// TIA Portal project "CompMC_TestProject" (V16)
// REr: Test project 1, RVS reiniging simpel

(* hardware
DEVICE "S71500/ET200MP station_1"  S7-1500 station
   slot 0: "Rail_0"  Rack  6ES7 590-1***0-0AA0
   slot 1: "PLC_1"  CPU 1513F-1 PN  6ES7 513-1FL02-0AB0  V2.8
      slot 3: "CPU display_1"  6ES7591-1AA00-0AA0
      slot 32768: "PROFINET interface_1"  X1
         slot 32769: "Port_1"  X1 P1
         slot 32770: "Port_2"  X1 P2
      slot 34817: "Virtual CP interface port_1"  Virtual CP interface port  Virtual CP interface port
   slot 2: "DI 16x24VDC / DQ 16x24VDC/0.5A BA_1"  DI 16x24VDC/DQ 16x24VDC/0.5A BA  6ES7 523-1BL00-0AA0  V1.1
*)

// ===== PLC "PLC_1"  CPU 1513F-1 PN =====

VAR_GLOBAL   // PLC tag table "Default tag table"
   "Tag_1" AT %M0.0 : Bool;
   "Var X" AT %MW100 : Word;
   "Alarm_1" AT %M102.0 : Bool;
   "Alarm_2" AT %M102.1 : Bool;
   "Alarm_3" AT %M102.2 : Bool;
   "Alarm_4" AT %M102.3 : Bool;
   "Result_as_Expected" AT %M103.0 : Bool;
   "X" AT %MW500 : Word;   // Variable X
   "Xnot10" AT %M400.0 : Bool;   // X != 10
   "Xnot12" AT %M400.1 : Bool;   // X != 12
   "Xnot15" AT %M400.2 : Bool;   // X != 15
   "Xnot20" AT %M400.3 : Bool;   // X != 20
   "NOK" AT %M400.7 : Bool;   // Result NOK
END_VAR

VAR_GLOBAL   // PLC tag table "InOut"
   "Ib_VlvLiq1Opened" AT %I0.0 : Bool;   // Valve liquid 1 openend
   "Ib_VlvLiq1Closed" AT %I0.1 : Bool;   // Valve liquid 1 closed
   "Ib_VlvLiq2Opened" AT %I0.2 : Bool;   // Valve liquid 2 opened
   "Ib_VlvLiq2Closed" AT %I0.3 : Bool;   // Valve liquid 2 closed
   "Ib_VlvDrnOpened" AT %I0.4 : Bool;   // Valve drain opened
   "Ib_VlvDrnClosed" AT %I0.5 : Bool;   // Valve drain closed
   "Ib_LvlContEmpty" AT %I0.6 : Bool;   // Level container empty
   "Ib_LvlContFull" AT %I0.7 : Bool;   // Level container full
   "Ib_PBFillLiq1" AT %I1.0 : Bool;   // Pushbutton fill container with liquid 1
   "Ib_PBFillLiq2" AT %I1.1 : Bool;   // Pushbutton fill container with liquid 2
   "Ib_PBEmptyCont" AT %I1.2 : Bool;   // Pushbutton empty container
   "Qb_VlvLiq1Open" AT %Q0.0 : Bool;   // Valve liquid 1 move open
   "Qb_VlvLiq2Open" AT %Q0.1 : Bool;   // Valve liquid 2 move open
   "Qb_VlvDrnOpen" AT %Q0.2 : Bool;   // Valve drain move open
   "Ib_PBStart" AT %I1.3 : Bool;   // Pushbutton start
   "Ib_PBStop" AT %I1.4 : Bool;   // Pushbutton stop
   "Ib_PBReset" AT %I1.5 : Bool;   // Pushbutton reset
END_VAR

VAR_GLOBAL CONSTANT   // PLC tag table "Open Library"
   "Modes.Auto" : Int := 1;
   "Modes.Manual" : Int := 2;
   "Modes.Independent" : Int := 10;
   "Modes.Stop" : Int := 0;
   "HMI.Status.Stopped" : Int := 0;
   "HMI.Status.Estop" : Int := 1;
   "HMI.Status.Error" : Int := 2;
   "HMI.Status.ForwardWork" : Int := 3;
   "HMI.Status.ReverseHome" : Int := 4;
   "HMI.Status.OnForwardWork" : Int := 5;
   "HMI.Status.OnReverseHome" : Int := 6;
   "IoScaling.S7Analog.Default.iRawMax" : Int := 27648;
   "IoScaling.S7Analog.Default.iRawMin" : Int := 0;
   "IoScaling.S7Analog.Default.bSwapBytes" : Bool := false;
   "IoScaling.S7Analog.+-V/mA.iRawMax" : Int := 27648;
   "IoScaling.S7Analog.+-V/mA.iRawMin" : Int := -27648;
   "IoScaling.S7Analog.Types.Default" : Int := 0;
   "IoScaling.S7Analog.Pt100.iRawMax" : Int := 8500;
   "IoScaling.S7Analog.Pt100.iRawMin" : Int := -2000;
   "IoScaling.S7Analog.Pt100.Climate.iRawMax" : Int := 13000;
   "IoScaling.S7Analog.Pt100.Climate.iRawMin" : Int := -12000;
   "IoScaling.S7Analog.Ni100.iRawMax" : Int := 2500;
   "IoScaling.S7Analog.Ni100.iRawMin" : Int := -600;
   "IoScaling.S7Analog.Ni100.Climate.iRawMax" : Int := 25000;
   "IoScaling.S7Analog.Ni100.Climate.iRawMin" : Int := -6000;
   "IoScaling.S7Analog.Types.+-V/mA" : Int := 1;
   "IoScaling.S7Analog.Types.Pt100" : Int := 2;
   "IoScaling.S7Analog.Types.Pt100.Climate" : Int := 3;
   "IoScaling.S7Analog.Types.Ni100" : Int := 4;
   "IoScaling.S7Analog.Types.Ni100.Climate" : Int := 5;
   "IoScaling.S7Analog.Pt100.rScaledMax" : Real := 850.0;
   "IoScaling.S7Analog.Pt100.rScaledMin" : Real := -200.0;
   "IoScaling.S7Analog.Pt100.Climate.rScaledMax" : Real := 130.0;
   "IoScaling.S7Analog.Pt100.Climate.rScaledMin" : Real := -120.0;
   "IoScaling.S7Analog.Ni100.rScaledMax" : Real := 250.0;
   "IoScaling.S7Analog.Ni100.rScaledMin" : Real := -60.0;
   "IoScaling.S7Analog.Ni100.Climate.rScaledMax" : Real := 250.0;
   "IoScaling.S7Analog.Ni100.Climate.rScaledMin" : Real := -60.0;
   "IoScaling.S7Analog.150Ohms.rScaledMax" : Real := 150.0;
   "IoScaling.S7Analog.150Ohms.rScaledMin" : Real := 0.0;
   "IoScaling.S7Analog.300Ohms.rScaledMax" : Real := 300.0;
   "IoScaling.S7Analog.300Ohms.rScaledMin" : Real := 0.0;
   "IoScaling.S7Analog.600Ohms.rScaledMax" : Real := 600.0;
   "IoScaling.S7Analog.600Ohms.rScaledMin" : Real := 0.0;
   "Estop.MinSetPoint" : Int := 0;
   "Estop.MaxSetPoint" : Int := 1;
   "Estop.HMISetPoint" : Int := 2;
   "Modes.PID.Inactive" : Int := 0;
   "Modes.PID.Pretuning" : Int := 1;
   "Modes.PID.FineTuning" : Int := 2;
   "Modes.PID.AutoMode" : Int := 3;
   "Modes.PID.ManualMode" : Int := 4;
   "HMI.Status.Generic1" : Int := 101;
   "HMI.Status.Generic2" : Int := 102;
   "HMI.Status.Generic3" : Int := 103;
   "HMI.Status.Generic4" : Int := 104;
   "HMI.Status.Generic5" : Int := 105;
   "HMI.Status.GenericNone" : Int := 100;
   "HMI.Status.Generic6" : Int := 106;
   "DataTypes.rMaxReal" : Real := 3.402823e38;
   "DataTypes.rMinReal" : Real := -3.402823e38;
   "DataTypes.iMaxInt" : Int := 32767;
   "DataTypes.iMinInt" : Int := -32768;
   "Handshakes.iSize" : Int := 5;
   "SoftStarter.Types.3RW30" : Int := 30;
   "SoftStarter.Types.3RW40" : Int := 40;
   "Simocode.Types.OverloadRelay" : Int := 0;
   "Simocode.Types.DirectStarter" : Int := 1;
   "Simocode.Types.ReversingStarter" : Int := 2;
   "SoftStarter.HMI.Status.RampDown" : Int := 5;
   "SoftStarter.HMI.Status.On" : Int := 4;
   "SoftStarter.HMI.Status.RampUp" : Int := 3;
   "SoftStarter.HMI.Status.EStop" : Int := 1;
   "SoftStarter.HMI.Status.Off" : Int := 0;
   "SoftStarter.HMI.Status.Error" : Int := 2;
   "FIFO.iQueueSize" : Int := 5;
   "FIFO.iQueueDisabled" : Int := -1;
   "TotalizerTimeUnits.MILLISECONDS" : Int := 0;
   "TotalizerTimeUnits.SECONDS" : Int := 1;
   "TotalizerTimeUnits.MINUTES" : Int := 2;
   "TotalizerTimeUnits.HOURS" : Int := 3;
   "TotalizerTimeUnits.DAYS" : Int := 4;
   "HMI.Status.SimulatedForwardWork" : Int := 7;
   "HMI.Status.SimulatedOnForwardWork" : Int := 9;
   "HMI.Status.SimulatedReverseHome" : Int := 8;
   "HMI.Status.SimulatedOnReverseHome" : Int := 10;
   "Ramp.Continuous" : Int := 0;
   "Ramp.Timed" : Int := 1;
END_VAR

// folder: Open Library V15/Data Types/Error

TYPE "udtError_Valve"
VERSION : 0.1
   STRUCT
      NoHomeFeedback : Bool;   // Home position feedback not active
      NoWorkFeedback : Bool;   // Work position feedback not active
      HomeFeedbackStillActive : Bool;   // Home position feedback still active
      WorkFeedbackStillActive : Bool;   // Work position feedback still active
   END_STRUCT;
END_TYPE

// folder: Open Library V15/Data Types/HMI

TYPE "udtHMI_ValveControl"
VERSION : 0.1
   STRUCT
      iMode : Int;   // Current mode
      iErrorCode : Int;   // Error code
      iStatus : Int;   // Status for HMI display
      bPB_ResetError : Bool;   // PB Reset block errors
      bPB_Home : Bool;   // PB Move to home in manual mode
      bPB_Work : Bool;   // PB Move to work in manual mode
      bPBEN_ResetError : Bool;   // PB Reset error enabled
      bPBEN_Home : Bool;   // PB Home enabled
      bPBEN_Work : Bool;   // PB Work enabled
      bHomeOn : Bool;   // Home command is on
      bWorkOn : Bool;   // Work command is on
      bSignalHome : Bool;   // Home feedback
      bSignalWork : Bool;   // Work feedback
      bError : Bool;   // Error status
      bInterlock : Bool;   // Valve interlocked
   END_STRUCT;
END_TYPE

// folder: (top level)

DATA_BLOCK "Program Logic_DB"   // DB2
{ S7_Optimized_Access := 'TRUE' }
VERSION : 0.1
// stored: InstanceOfName Program Logic
"Program Logic"
BEGIN
END_DATA_BLOCK

DATA_BLOCK "DB_HMI"   // DB3
{ S7_Optimized_Access := 'TRUE' }
VERSION : 0.1
   VAR
      VlvLiq1 : "udtHMI_ValveControl";
      VlvLiq2 : "udtHMI_ValveControl";
      VlvDrn : "udtHMI_ValveControl";
   END_VAR
BEGIN
END_DATA_BLOCK

DATA_BLOCK "DB_ProgramLogic"   // DB4
{ S7_Optimized_Access := 'TRUE' }
VERSION : 0.1
   VAR
      VlvLiq1_Open : Bool;
      VlvLiq2_Open : Bool;
      VlvDrn_Open : Bool;
   END_VAR
BEGIN
END_DATA_BLOCK

DATA_BLOCK "Valve Drain_DB"   // DB7
{ S7_Optimized_Access := 'TRUE' }
VERSION : 0.1
// stored: InstanceOfName Valve Drain
"Valve Drain"
BEGIN
END_DATA_BLOCK

DATA_BLOCK "Valve Liquid 1_DB"   // DB8
{ S7_Optimized_Access := 'TRUE' }
VERSION : 0.1
// stored: InstanceOfName Valve Liquid 1
"Valve Liquid 1"
BEGIN
END_DATA_BLOCK

DATA_BLOCK "Valve Liquid 2_DB"   // DB9
{ S7_Optimized_Access := 'TRUE' }
VERSION : 0.1
// stored: InstanceOfName Valve Liquid 2
"Valve Liquid 2"
BEGIN
END_DATA_BLOCK

FUNCTION_BLOCK "Valve Liquid 1"   // FB2, FBD
{ S7_Optimized_Access := 'TRUE' }
VERSION : 0.1
   VAR
      VlvLiq1 : "fbValve_Solenoid";
   END_VAR
BEGIN

REGION Network 1
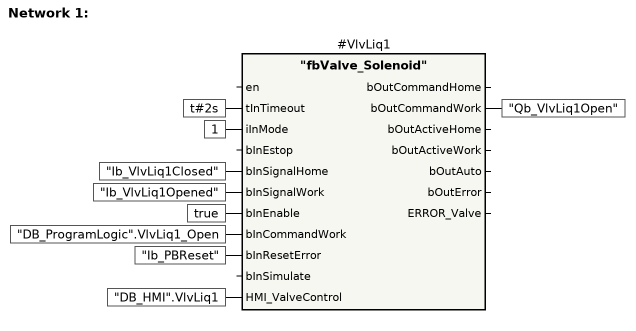
   #VlvLiq1(tInTimeout := t#2s,   // "fbValve_Solenoid"
            iInMode := 1,
            bInSignalHome := "Ib_VlvLiq1Closed",
            bInSignalWork := "Ib_VlvLiq1Opened",
            bInEnable := true,
            bInCommandWork := "DB_ProgramLogic".VlvLiq1_Open,
            bInResetError := "Ib_PBReset",
            HMI_ValveControl := "DB_HMI".VlvLiq1,
            bOutCommandWork => "Qb_VlvLiq1Open");
END_REGION
END_FUNCTION_BLOCK

FUNCTION_BLOCK "Valve Liquid 2"   // FB3, FBD
{ S7_Optimized_Access := 'TRUE' }
VERSION : 0.1
   VAR
      VlvLiq2 : "fbValve_Solenoid";
   END_VAR
BEGIN

REGION Network 1
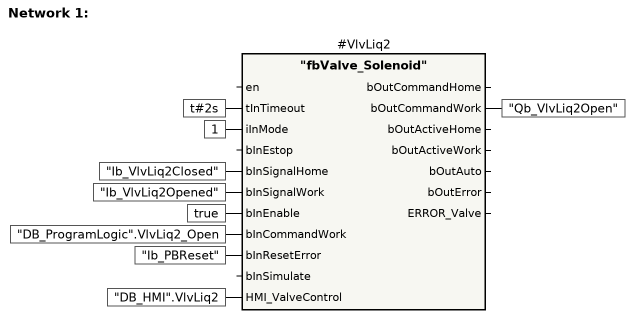
   #VlvLiq2(tInTimeout := t#2s,   // "fbValve_Solenoid"
            iInMode := 1,
            bInSignalHome := "Ib_VlvLiq2Closed",
            bInSignalWork := "Ib_VlvLiq2Opened",
            bInEnable := true,
            bInCommandWork := "DB_ProgramLogic".VlvLiq2_Open,
            bInResetError := "Ib_PBReset",
            HMI_ValveControl := "DB_HMI".VlvLiq2,
            bOutCommandWork => "Qb_VlvLiq2Open");
END_REGION
END_FUNCTION_BLOCK

FUNCTION_BLOCK "Valve Drain"   // FB4, FBD
{ S7_Optimized_Access := 'TRUE' }
VERSION : 0.1
   VAR
      VlvDrn : "fbValve_Solenoid";
   END_VAR
BEGIN

REGION Network 1
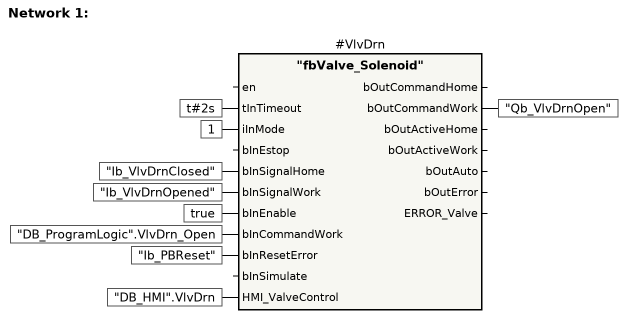
   #VlvDrn(tInTimeout := t#2s,   // "fbValve_Solenoid"
           iInMode := 1,
           bInSignalHome := "Ib_VlvDrnClosed",
           bInSignalWork := "Ib_VlvDrnOpened",
           bInEnable := true,
           bInCommandWork := "DB_ProgramLogic".VlvDrn_Open,
           bInResetError := "Ib_PBReset",
           HMI_ValveControl := "DB_HMI".VlvDrn,
           bOutCommandWork => "Qb_VlvDrnOpen");
END_REGION
END_FUNCTION_BLOCK

FUNCTION_BLOCK "Program Logic"   // FB5, FBD
{ S7_Optimized_Access := 'TRUE' }
VERSION : 0.1
   VAR
      StepSeq : "fbStepSequencer";
      CurrentStep : Int;
      NextStep : Int;
      StepDone : Bool;
   END_VAR
   VAR_TEMP   // added for the SCL form of the ladder/FBD networks
      _w1 : Bool;
   END_VAR
BEGIN

REGION Network 1: 0 -- Idle
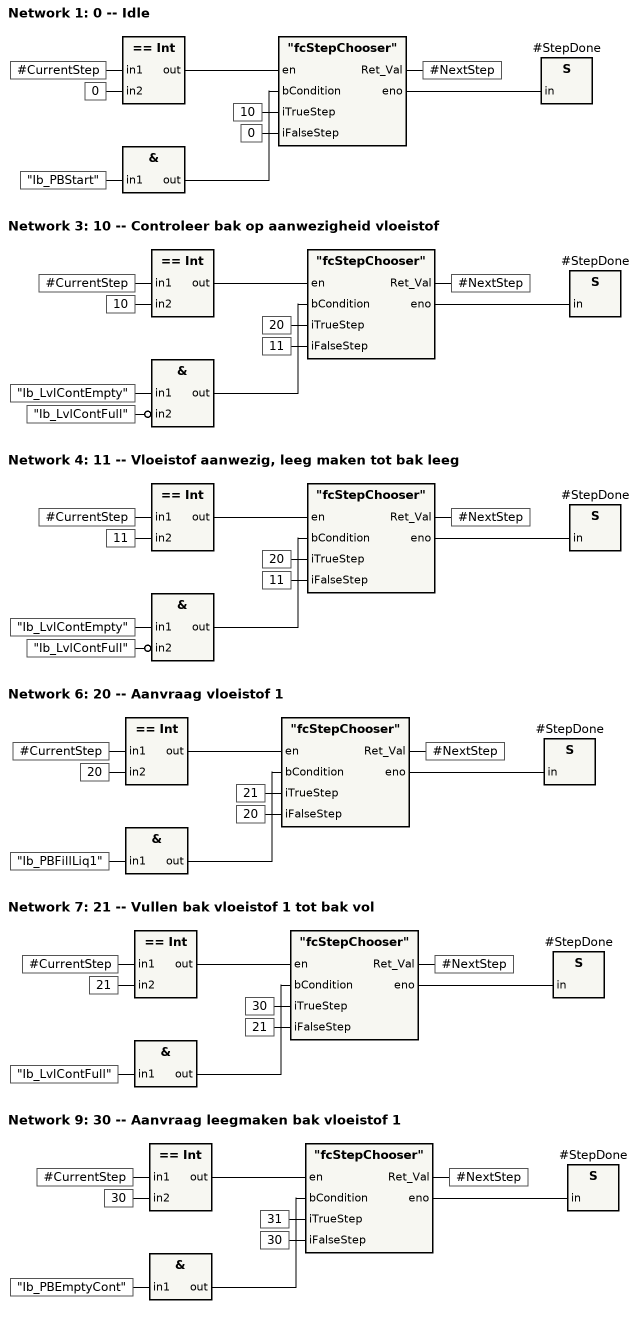
   #NextStep := "fcStepChooser"(EN := #CurrentStep = 0,
                           bCondition := "Ib_PBStart",
                           iTrueStep := 10,
                           iFalseStep := 0,
                           ENO => #_w1);
   IF #_w1 THEN #StepDone := TRUE; END_IF;
END_REGION

REGION Network 3: 10 -- Controleer bak op aanwezigheid vloeistof
   // vloeistof aanwezig 10->11
   // geen vloeistof aanwezig 10->20
   #NextStep := "fcStepChooser"(EN := #CurrentStep = 10,
                           bCondition := "Ib_LvlContEmpty" AND NOT "Ib_LvlContFull",
                           iTrueStep := 20,
                           iFalseStep := 11,
                           ENO => #_w1);
   IF #_w1 THEN #StepDone := TRUE; END_IF;
END_REGION

REGION Network 4: 11 -- Vloeistof aanwezig, leeg maken tot bak leeg
   #NextStep := "fcStepChooser"(EN := #CurrentStep = 11,
                           bCondition := "Ib_LvlContEmpty" AND NOT "Ib_LvlContFull",
                           iTrueStep := 20,
                           iFalseStep := 11,
                           ENO => #_w1);
   IF #_w1 THEN #StepDone := TRUE; END_IF;
END_REGION

REGION Network 6: 20 -- Aanvraag vloeistof 1
   #NextStep := "fcStepChooser"(EN := #CurrentStep = 20,
                           bCondition := "Ib_PBFillLiq1",
                           iTrueStep := 21,
                           iFalseStep := 20,
                           ENO => #_w1);
   IF #_w1 THEN #StepDone := TRUE; END_IF;
END_REGION

REGION Network 7: 21 -- Vullen bak vloeistof 1 tot bak vol
   #NextStep := "fcStepChooser"(EN := #CurrentStep = 21,
                           bCondition := "Ib_LvlContFull",
                           iTrueStep := 30,
                           iFalseStep := 21,
                           ENO => #_w1);
   IF #_w1 THEN #StepDone := TRUE; END_IF;
END_REGION

REGION Network 9: 30 -- Aanvraag leegmaken bak vloeistof 1
   #NextStep := "fcStepChooser"(EN := #CurrentStep = 30,
                           bCondition := "Ib_PBEmptyCont",
                           iTrueStep := 31,
                           iFalseStep := 30,
                           ENO => #_w1);
   IF #_w1 THEN #StepDone := TRUE; END_IF;
END_REGION

REGION Network 10: 31 -- Leeg maken bak vloeistof 1
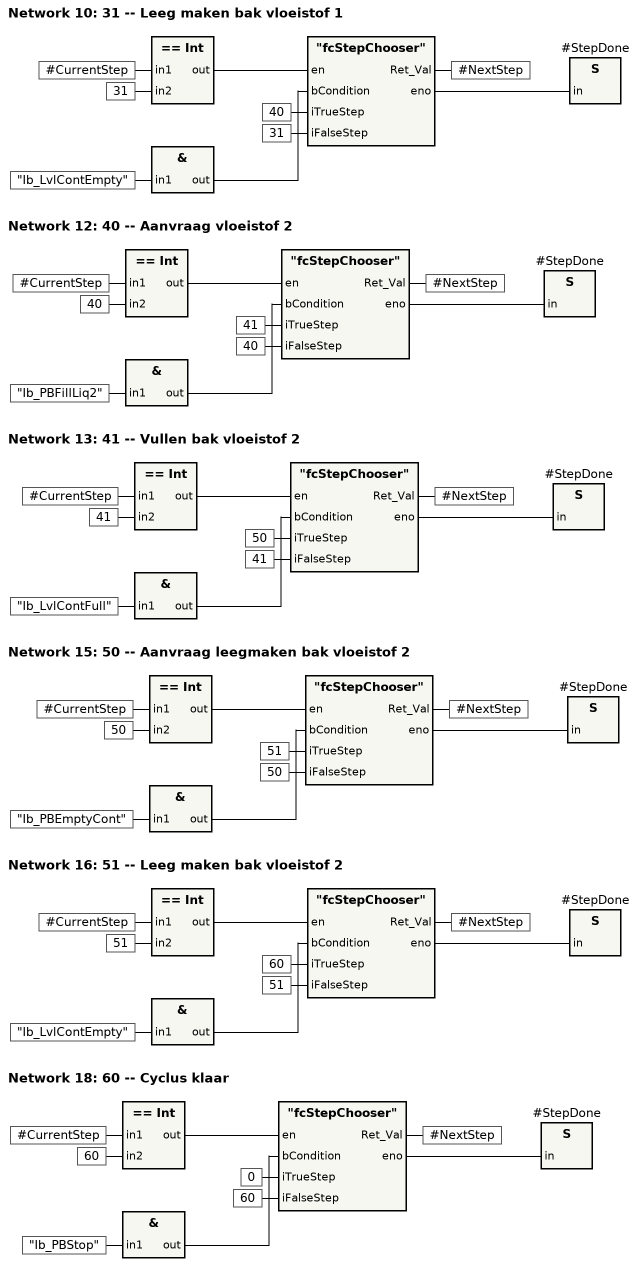
   #NextStep := "fcStepChooser"(EN := #CurrentStep = 31,
                           bCondition := "Ib_LvlContEmpty",
                           iTrueStep := 40,
                           iFalseStep := 31,
                           ENO => #_w1);
   IF #_w1 THEN #StepDone := TRUE; END_IF;
END_REGION

REGION Network 12: 40 -- Aanvraag vloeistof 2
   #NextStep := "fcStepChooser"(EN := #CurrentStep = 40,
                           bCondition := "Ib_PBFillLiq2",
                           iTrueStep := 41,
                           iFalseStep := 40,
                           ENO => #_w1);
   IF #_w1 THEN #StepDone := TRUE; END_IF;
END_REGION

REGION Network 13: 41 -- Vullen bak vloeistof 2
   #NextStep := "fcStepChooser"(EN := #CurrentStep = 41,
                           bCondition := "Ib_LvlContFull",
                           iTrueStep := 50,
                           iFalseStep := 41,
                           ENO => #_w1);
   IF #_w1 THEN #StepDone := TRUE; END_IF;
END_REGION

REGION Network 15: 50 -- Aanvraag leegmaken bak vloeistof 2
   #NextStep := "fcStepChooser"(EN := #CurrentStep = 50,
                           bCondition := "Ib_PBEmptyCont",
                           iTrueStep := 51,
                           iFalseStep := 50,
                           ENO => #_w1);
   IF #_w1 THEN #StepDone := TRUE; END_IF;
END_REGION

REGION Network 16: 51 -- Leeg maken bak vloeistof 2
   #NextStep := "fcStepChooser"(EN := #CurrentStep = 51,
                           bCondition := "Ib_LvlContEmpty",
                           iTrueStep := 60,
                           iFalseStep := 51,
                           ENO => #_w1);
   IF #_w1 THEN #StepDone := TRUE; END_IF;
END_REGION

REGION Network 18: 60 -- Cyclus klaar
   #NextStep := "fcStepChooser"(EN := #CurrentStep = 60,
                           bCondition := "Ib_PBStop",
                           iTrueStep := 0,
                           iFalseStep := 60,
                           ENO => #_w1);
   IF #_w1 THEN #StepDone := TRUE; END_IF;
END_REGION

REGION Network 20: Step Sequencer
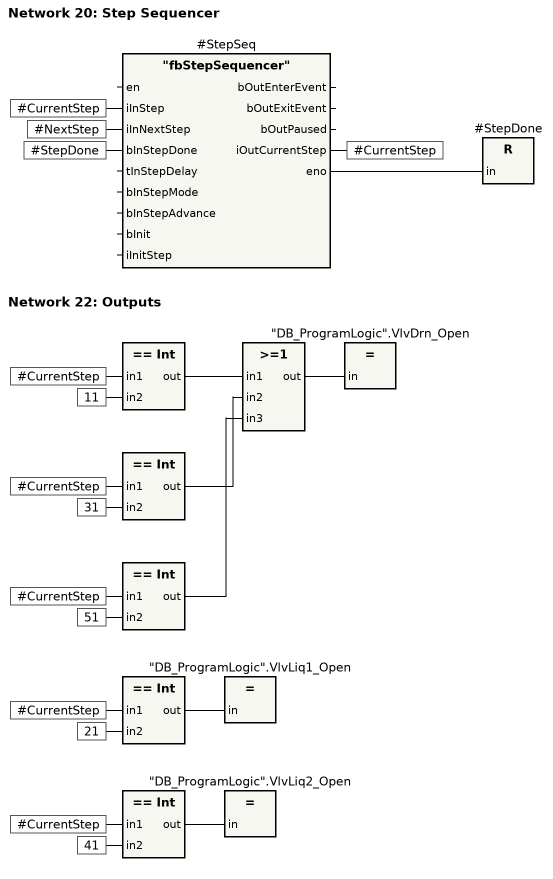
   #StepSeq(iInStep := #CurrentStep,   // "fbStepSequencer"
            iInNextStep := #NextStep,
            bInStepDone := #StepDone,
            iOutCurrentStep => #CurrentStep,
            ENO => #_w1);
   IF #_w1 THEN #StepDone := FALSE; END_IF;
END_REGION

REGION Network 22: Outputs
   "DB_ProgramLogic".VlvDrn_Open := (#CurrentStep = 11) OR (#CurrentStep = 31) OR (#CurrentStep = 51);
   "DB_ProgramLogic".VlvLiq1_Open := #CurrentStep = 21;
   "DB_ProgramLogic".VlvLiq2_Open := #CurrentStep = 41;
END_REGION
END_FUNCTION_BLOCK

ORGANIZATION_BLOCK "Main"   // OB1, FBD, ProgramCycle
TITLE = "Main Program Sweep (Cycle)"
{ S7_Optimized_Access := 'TRUE' }
VERSION : 0.1
   VAR_INPUT
      Initial_Call : Bool;   // Initial call of this OB
      Remanence : Bool;   // =True, if remanent data are available
   END_VAR
BEGIN

REGION Network 1
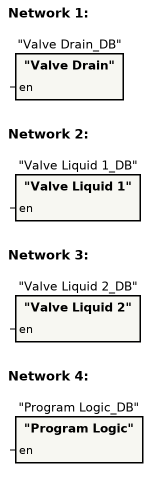
   "Valve Drain_DB"();   // "Valve Drain"
END_REGION

REGION Network 2
   "Valve Liquid 1_DB"();   // "Valve Liquid 1"
END_REGION

REGION Network 3
   "Valve Liquid 2_DB"();   // "Valve Liquid 2"
END_REGION

REGION Network 4
   "Program Logic_DB"();   // "Program Logic"
END_REGION
END_ORGANIZATION_BLOCK

// folder: Open Library V15/Devices

FUNCTION_BLOCK "fbValve_Solenoid"   // FB110, FBD
TITLE = Controls a double- or single-acting valve
{ S7_Optimized_Access := 'TRUE' }
VERSION : 0.1
   VAR_INPUT
      tInTimeout : Time;   // Timeout time for an actuator's feedback to activate before giving a fault
      iInMode : Int;   // Mode Selection
      bInEstop : Bool;   // Estop
      bInSignalHome : Bool;   // Home position feedback
      bInSignalWork : Bool;   // Work position feedback
      bInEnable : Bool;   // Home and Work Enabled
      bInCommandWork : Bool;   // Move to work position in automatic mode
      bInResetError : Bool;   // Reset Error
      bInSimulate : Bool;   // Activate device simulation
   END_VAR
   VAR_OUTPUT
      bOutCommandHome : Bool;   // Home position command
      bOutCommandWork : Bool;   // Work position command
      bOutActiveHome : Bool;   // Valve is in home position
      bOutActiveWork : Bool;   // Valve is in work position
      bOutAuto : Bool;   // Block in auto mode
      bOutError : Bool;   // Error exists
      ERROR_Valve : "udtError_Valve";   // Valve error structure
   END_VAR
   VAR_IN_OUT
      HMI_ValveControl : "udtHMI_ValveControl";   // HMI valve control
   END_VAR
   VAR
      ErrorScroller : "fbErrorScroller";   // Sub-block to handle error scroller
      TON_TimeOut : TON_TIME;   // Timer for Error Timeout
      iLastMode : Int;   // Last mode code
      bNewMode : Bool;   // New mode selected
      bEnableHome : Bool;   // Home position enabled
      bEnableWork : Bool;   // Work position enabled
      bAutoMode : Bool;   // Auto Mode is active
      bManualMode : Bool;   // Manual Mode is active
      bReset : Bool;
      bTON_TimeOut : Bool;
      bPB_Home : Bool;
      bPB_Work : Bool;
      bPB_ResetError : Bool;
   END_VAR
   VAR_TEMP
      tTimeoutElapsed : Time;   // Elapsed time for TON_Timeout
      bTemp : Bool;
   END_VAR
   VAR_TEMP   // added for the SCL form of the ladder/FBD networks
      _w1 : Bool;
      _w2 : Bool;
   END_VAR
BEGIN

REGION Network 1: --------------------------------------------------------- Inputs ------------------------------------------------------------------
END_REGION

REGION Network 2: Read HMI input buttons
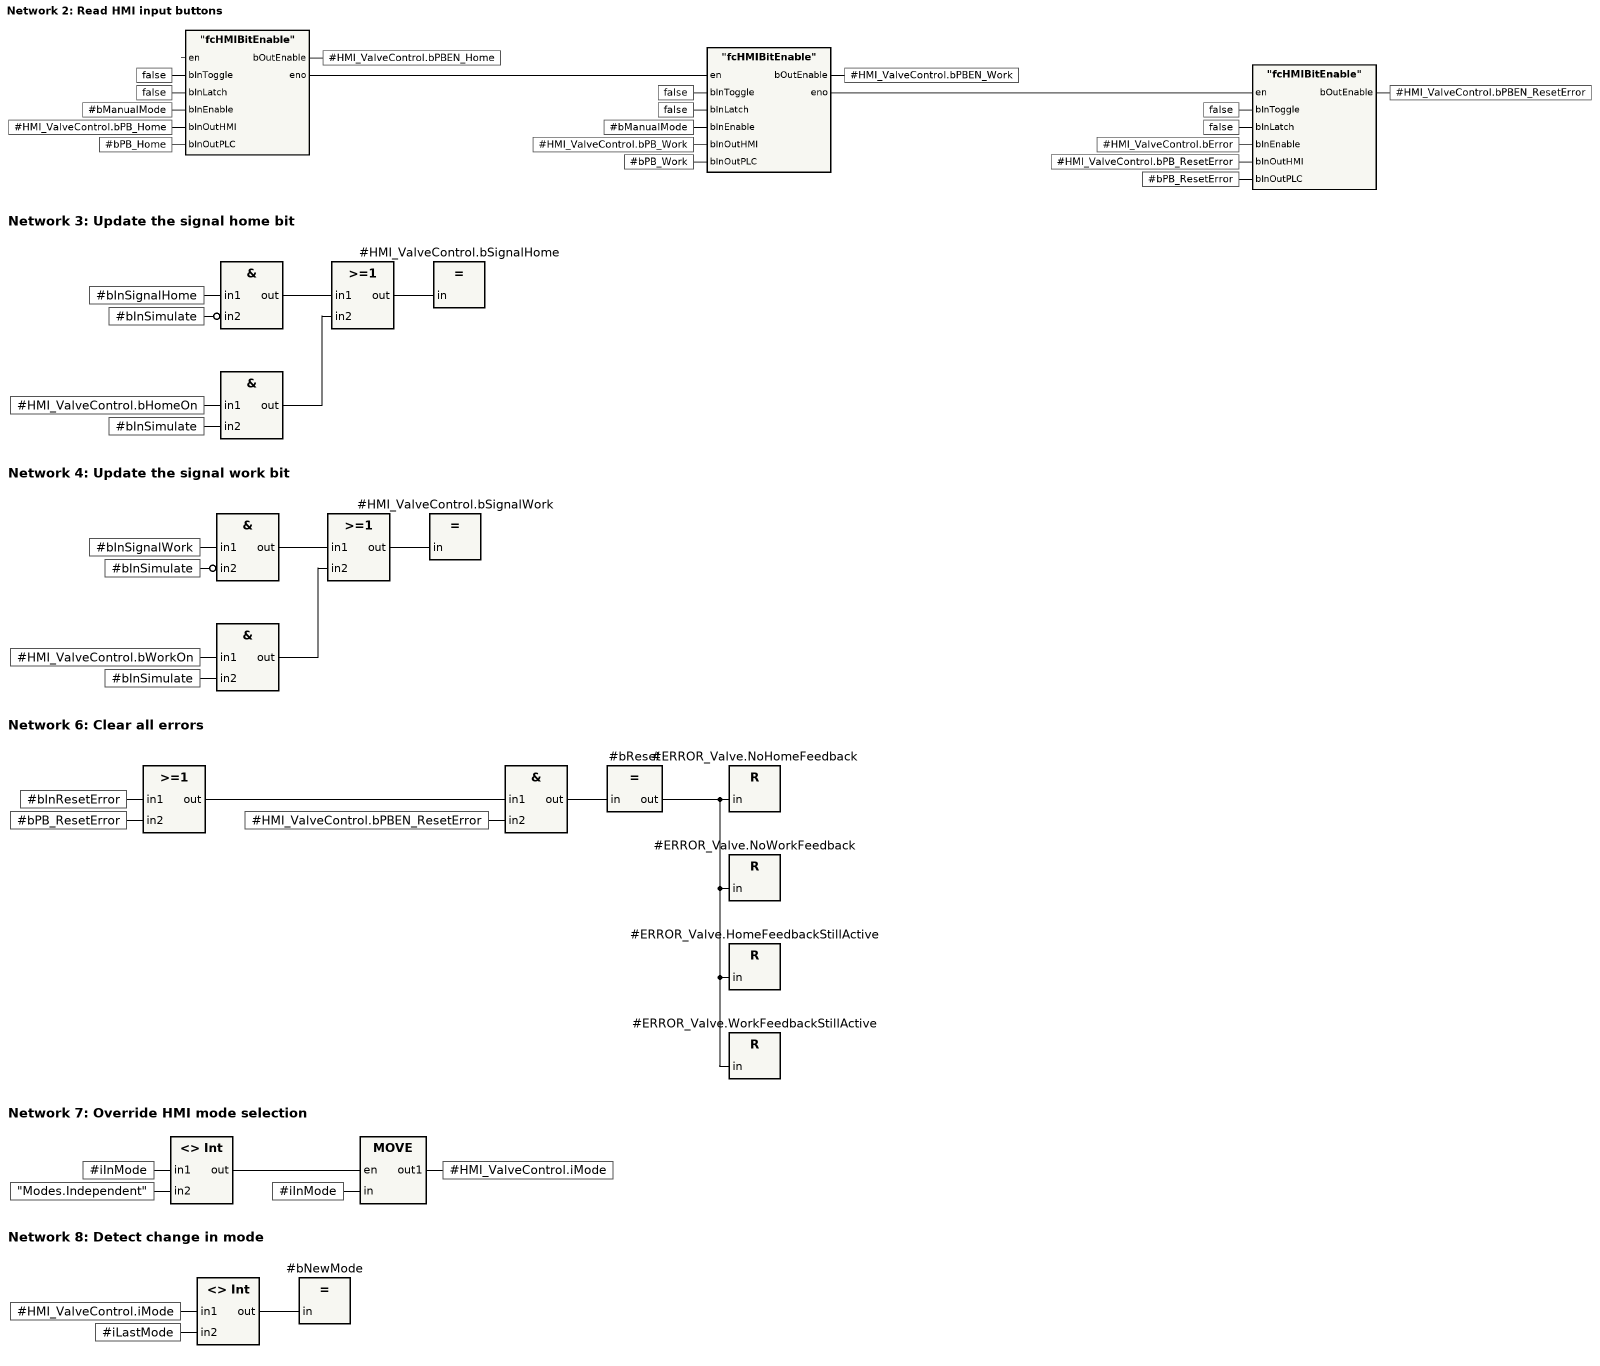
   "fcHMIBitEnable"(bInToggle := false,
                    bInLatch := false,
                    bInEnable := #bManualMode,
                    bInOutHMI := #HMI_ValveControl.bPB_Home,
                    bInOutPLC := #bPB_Home,
                    bOutEnable => #HMI_ValveControl.bPBEN_Home,
                    ENO => #_w1);
   "fcHMIBitEnable"(EN := #_w1,
                    bInToggle := false,
                    bInLatch := false,
                    bInEnable := #bManualMode,
                    bInOutHMI := #HMI_ValveControl.bPB_Work,
                    bInOutPLC := #bPB_Work,
                    bOutEnable => #HMI_ValveControl.bPBEN_Work,
                    ENO => #_w2);
   IF #_w2 THEN
       "fcHMIBitEnable"(bInToggle := false,
                        bInLatch := false,
                        bInEnable := #HMI_ValveControl.bError,
                        bInOutHMI := #HMI_ValveControl.bPB_ResetError,
                        bInOutPLC := #bPB_ResetError,
                        bOutEnable => #HMI_ValveControl.bPBEN_ResetError);
   END_IF;
END_REGION

REGION Network 3: Update the signal home bit
   #HMI_ValveControl.bSignalHome := (#bInSignalHome AND NOT #bInSimulate) OR (#HMI_ValveControl.bHomeOn AND #bInSimulate);
END_REGION

REGION Network 4: Update the signal work bit
   #HMI_ValveControl.bSignalWork := (#bInSignalWork AND NOT #bInSimulate) OR (#HMI_ValveControl.bWorkOn AND #bInSimulate);
END_REGION

REGION Network 5: --------------------------------------------------- Control Logic ------------------------------------------------------------
END_REGION

REGION Network 6: Clear all errors
   #bReset := (#bInResetError OR #bPB_ResetError) AND #HMI_ValveControl.bPBEN_ResetError;
   IF #bReset THEN
       #ERROR_Valve.NoHomeFeedback := FALSE;
       #ERROR_Valve.NoWorkFeedback := FALSE;
       #ERROR_Valve.HomeFeedbackStillActive := FALSE;
       #ERROR_Valve.WorkFeedbackStillActive := FALSE;
   END_IF;
END_REGION

REGION Network 7: Override HMI mode selection
   IF #iInMode <> "Modes.Independent" THEN #HMI_ValveControl.iMode := #iInMode; END_IF;
END_REGION

REGION Network 8: Detect change in mode
   #bNewMode := #HMI_ValveControl.iMode <> #iLastMode;
END_REGION

REGION Network 9: Keep track of last mode
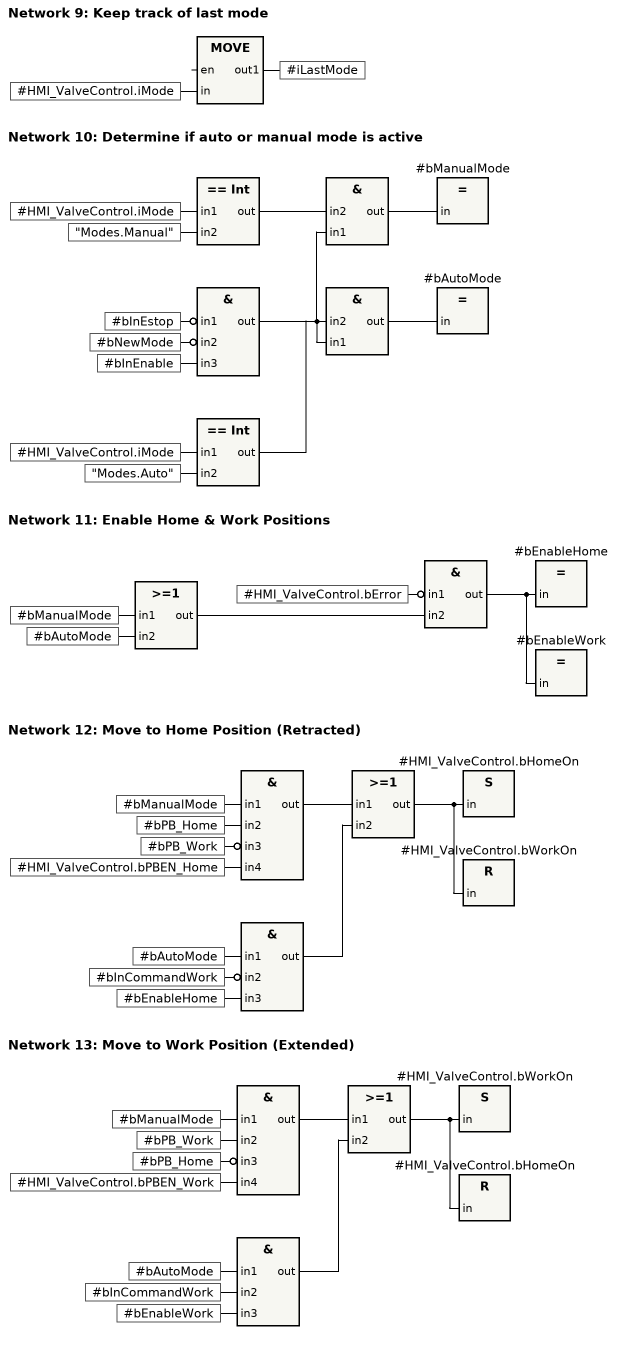
   #iLastMode := #HMI_ValveControl.iMode;
END_REGION

REGION Network 10: Determine if auto or manual mode is active
   #_w1 := NOT #bInEstop AND NOT #bNewMode AND #bInEnable;
   #bManualMode := (#HMI_ValveControl.iMode = "Modes.Manual") AND #_w1;
   #bAutoMode := (#HMI_ValveControl.iMode = "Modes.Auto") AND #_w1;
END_REGION

REGION Network 11: Enable Home & Work Positions
   // IF manual mode AND no estop AND not a new mode AND enabled => 
   // --if no cylinder errors, enable move to Home and Work
   // --enable home and work HMI buttons only in manual mode
   #bEnableHome := NOT #HMI_ValveControl.bError AND (#bManualMode OR #bAutoMode);
   #bEnableWork := #bEnableHome;
END_REGION

REGION Network 12: Move to Home Position (Retracted)
   // IF manual mode and home button is pressed =>
   // --Set close cylinder
   IF (#bManualMode AND #bPB_Home AND NOT #bPB_Work AND #HMI_ValveControl.bPBEN_Home) OR (#bAutoMode AND NOT #bInCommandWork AND #bEnableHome) THEN
       #HMI_ValveControl.bHomeOn := TRUE;
       #HMI_ValveControl.bWorkOn := FALSE;
   END_IF;
END_REGION

REGION Network 13: Move to Work Position (Extended)
   // IF manual mode and work button button is pressed =>
   // --Set open cylinder
   IF (#bManualMode AND #bPB_Work AND NOT #bPB_Home AND #HMI_ValveControl.bPBEN_Work) OR (#bAutoMode AND #bInCommandWork AND #bEnableWork) THEN
       #HMI_ValveControl.bWorkOn := TRUE;
       #HMI_ValveControl.bHomeOn := FALSE;
   END_IF;
END_REGION

REGION Network 14: Reset home on if not enabled
   // IF in auto AND home is not enabled => RESET home command
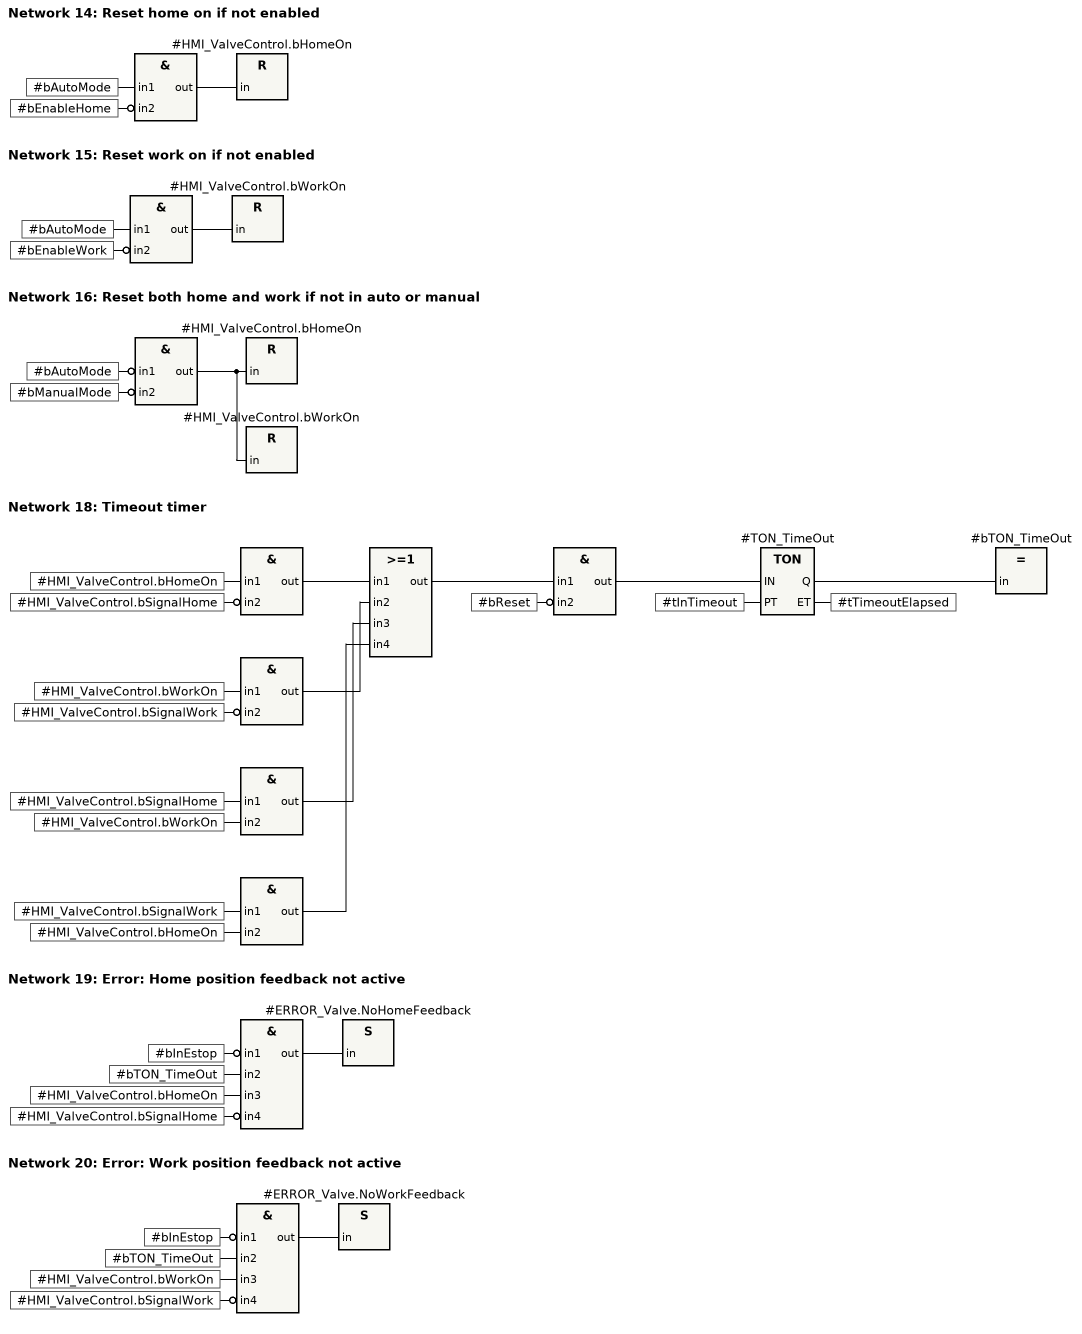
   IF #bAutoMode AND NOT #bEnableHome THEN #HMI_ValveControl.bHomeOn := FALSE; END_IF;
END_REGION

REGION Network 15: Reset work on if not enabled
   // IF in auto AND work is not enabled => RESET work command
   IF #bAutoMode AND NOT #bEnableWork THEN #HMI_ValveControl.bWorkOn := FALSE; END_IF;
END_REGION

REGION Network 16: Reset both home and work if not in auto or manual
   // IF not in auto AND not in manual => RESET home and work commands
   IF NOT #bAutoMode AND NOT #bManualMode THEN
       #HMI_ValveControl.bHomeOn := FALSE;
       #HMI_ValveControl.bWorkOn := FALSE;
   END_IF;
END_REGION

REGION Network 17: --------------------------------------------------------- Errors ------------------------------------------------------------------
END_REGION

REGION Network 18: Timeout timer
   // Time delay for errors
   #TON_TimeOut(IN := ((#HMI_ValveControl.bHomeOn AND NOT #HMI_ValveControl.bSignalHome) OR (#HMI_ValveControl.bWorkOn AND NOT #HMI_ValveControl.bSignalWork) OR (#HMI_ValveControl.bSignalHome AND #HMI_ValveControl.bWorkOn) OR (#HMI_ValveControl.bSignalWork AND #HMI_ValveControl.bHomeOn)) AND NOT #bReset,   // TON
                PT := #tInTimeout,
                ET => #tTimeoutElapsed);
   #bTON_TimeOut := #TON_TimeOut.Q;
END_REGION

REGION Network 19: Error: Home position feedback not active
   IF NOT #bInEstop AND #bTON_TimeOut AND #HMI_ValveControl.bHomeOn AND NOT #HMI_ValveControl.bSignalHome THEN
       #ERROR_Valve.NoHomeFeedback := TRUE;
   END_IF;
END_REGION

REGION Network 20: Error: Work position feedback not active
   // Not reach work position
   IF NOT #bInEstop AND #bTON_TimeOut AND #HMI_ValveControl.bWorkOn AND NOT #HMI_ValveControl.bSignalWork THEN
       #ERROR_Valve.NoWorkFeedback := TRUE;
   END_IF;
END_REGION

REGION Network 21: Error: Home position feedback still active
   // Home position still active
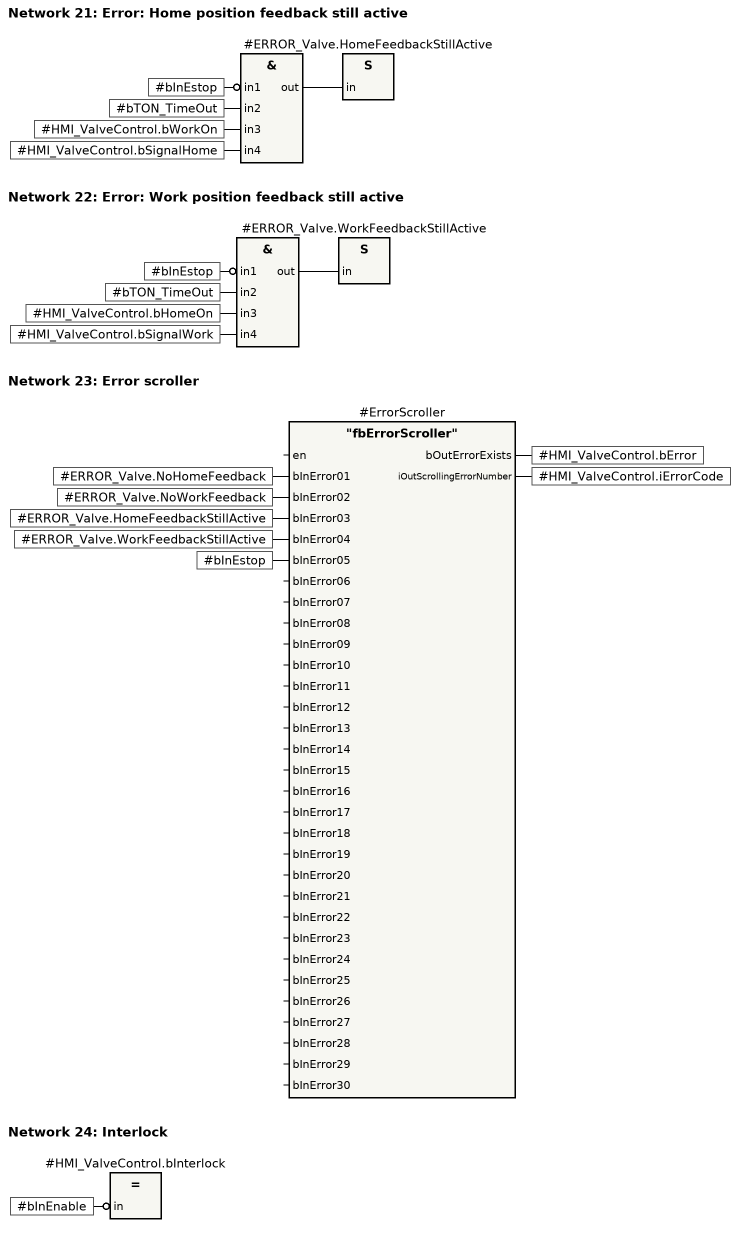
   IF NOT #bInEstop AND #bTON_TimeOut AND #HMI_ValveControl.bWorkOn AND #HMI_ValveControl.bSignalHome THEN
       #ERROR_Valve.HomeFeedbackStillActive := TRUE;
   END_IF;
END_REGION

REGION Network 22: Error: Work position feedback still active
   // Work position still active
   IF NOT #bInEstop AND #bTON_TimeOut AND #HMI_ValveControl.bHomeOn AND #HMI_ValveControl.bSignalWork THEN
       #ERROR_Valve.WorkFeedbackStillActive := TRUE;
   END_IF;
END_REGION

REGION Network 23: Error scroller
   // Call the Error-Scroller which cyles through all possible errors and checks 
   // their state for display on the HMI
   #ErrorScroller(bInError01 := #ERROR_Valve.NoHomeFeedback,   // "fbErrorScroller"
                  bInError02 := #ERROR_Valve.NoWorkFeedback,
                  bInError03 := #ERROR_Valve.HomeFeedbackStillActive,
                  bInError04 := #ERROR_Valve.WorkFeedbackStillActive,
                  bInError05 := #bInEstop,
                  bOutErrorExists => #HMI_ValveControl.bError,
                  iOutScrollingErrorNumber => #HMI_ValveControl.iErrorCode);
END_REGION

REGION Network 24: Interlock
   #HMI_ValveControl.bInterlock := NOT #bInEnable;
END_REGION

REGION Network 25: Set HMI status
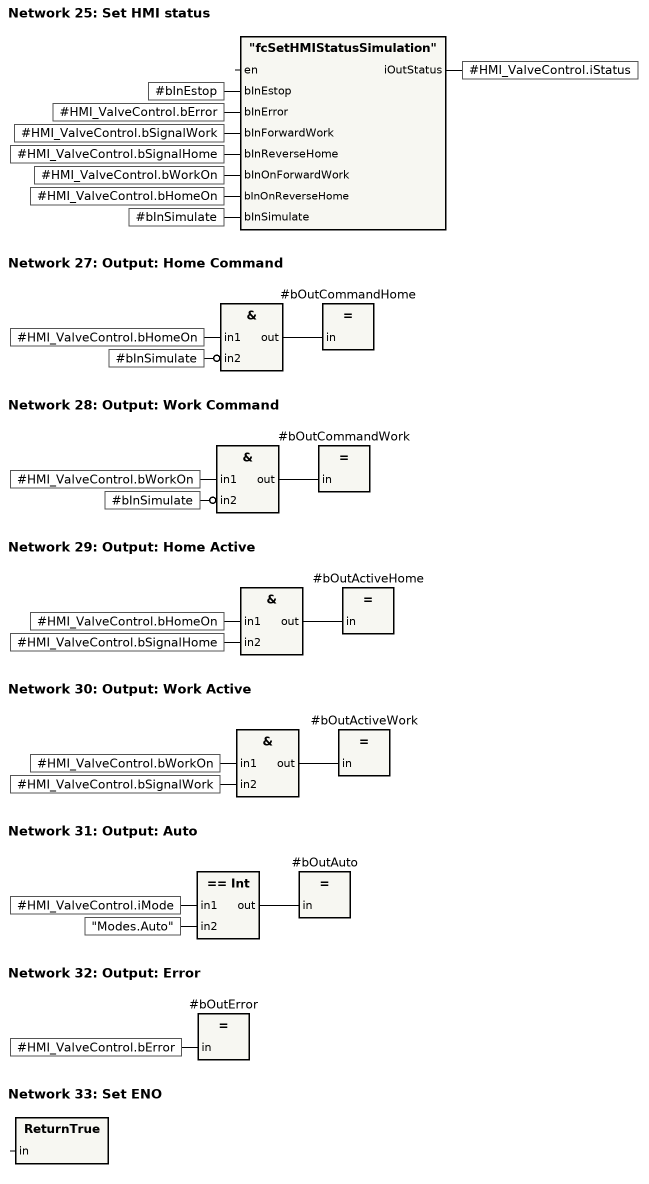
   "fcSetHMIStatusSimulation"(bInEstop := #bInEstop,
                           bInError := #HMI_ValveControl.bError,
                           bInForwardWork := #HMI_ValveControl.bSignalWork,
                           bInReverseHome := #HMI_ValveControl.bSignalHome,
                           bInOnForwardWork := #HMI_ValveControl.bWorkOn,
                           bInOnReverseHome := #HMI_ValveControl.bHomeOn,
                           bInSimulate := #bInSimulate,
                           iOutStatus => #HMI_ValveControl.iStatus);
END_REGION

REGION Network 26: -------------------------------------------------- Outputs --------------------------------------------------
END_REGION

REGION Network 27: Output: Home Command
   #bOutCommandHome := #HMI_ValveControl.bHomeOn AND NOT #bInSimulate;
END_REGION

REGION Network 28: Output: Work Command
   #bOutCommandWork := #HMI_ValveControl.bWorkOn AND NOT #bInSimulate;
END_REGION

REGION Network 29: Output: Home Active
   #bOutActiveHome := #HMI_ValveControl.bHomeOn AND #HMI_ValveControl.bSignalHome;
END_REGION

REGION Network 30: Output: Work Active
   #bOutActiveWork := #HMI_ValveControl.bWorkOn AND #HMI_ValveControl.bSignalWork;
END_REGION

REGION Network 31: Output: Auto
   #bOutAuto := #HMI_ValveControl.iMode = "Modes.Auto";
END_REGION

REGION Network 32: Output: Error
   #bOutError := #HMI_ValveControl.bError;
END_REGION

REGION Network 33: Set ENO
   ENO := TRUE;
   RETURN;
END_REGION
END_FUNCTION_BLOCK

// folder: Open Library V15/Process

FUNCTION_BLOCK "fbStepSequencer"   // FB185, SCL
TITLE = Step sequence controller
{ S7_Optimized_Access := 'TRUE' }
AUTHOR : Boris
VERSION : 4.0
// Modified by Ken Brey 2010-08-25 KLB.  Added Initialization inputs and logic.
// Modified by Ken Brey 2006-08-08 Removed initialization of inputs.  Initializing inputs doesn't do anything.  The input value if un-wired will be the last value
//                                   set for that input in a different call.  The initialized value in the declaration section does not set it back to default
//                                   if unwired.  Allways supply values for all inputs.
// Modified by Tim Jager 2005-12-13 no block Id in error message
// Modified by Boris: branched -> simplified version, no errors, no timeout; still have to use static memory for TON/CurStep (might be fixed later using in/out structure)
// Modified by Nick Shea:  2012-03-30 Re-instated step mode
   VAR_INPUT
      iInStep : Int;   // Constant: current step required for the FB to run
      iInNextStep : Int;   // Next step to go to if step is done
      bInStepDone : Bool;   // if step done logic is true, then we move from IN_STEP to NEXT_STEP
      tInStepDelay : Time;   // After the step done input is true, we wait for x seconds before moving to next
      bInStepMode : Bool;   // Pause sequence at completion of current step
      bInStepAdvance : Bool;   // If paused, trigger next step
      bInit : Bool;
      iInitStep : Int;
   END_VAR
   VAR_OUTPUT
      bOutEnterEvent : Bool;
      bOutExitEvent : Bool;
      bOutPaused : Bool;   // Sequence is currently paused.
      iOutCurrentStep : Int;   // output current step
   END_VAR
   VAR
      TON_StepDelay : TON_TIME;   // used to delay moving to the next step.
      iCurrentStep : Int;   // Current step of the sequencer
      bAlreadyInThisStep : Bool;
   END_VAR
   VAR_TEMP
      bNoStepDelay : Bool;   // step delay disabled
   END_VAR
BEGIN


   //*****************************************************************************************
   // INSTRUCTION SECTION
   ENO:=false; //init variables
   #bOutExitEvent :=false;
   #bOutEnterEvent:=false;

   IF (#iInStep=#iCurrentStep) THEN
       IF NOT #bAlreadyInThisStep THEN
           #bOutEnterEvent:=true;
           #bAlreadyInThisStep:=true;
       END_IF;
       IF #bInStepDone THEN
           //Run Step done Timer
           #TON_StepDelay(IN:=(TRUE),PT:=#tInStepDelay);

           //check if we are using a step delay
           #bNoStepDelay:= (#tInStepDelay<=T#0MS);

           //We can move to the next step if (STEP_DONE and StepDelay timer complete) 
           //  AND
           //(we are in step mode and the step advance is true, or if we are not in step mode 
           //  AND
           //It is not the first scan of this step
           IF ((#TON_StepDelay.Q OR #bNoStepDelay) AND (NOT #bInStepMode OR (#bInStepMode AND #bInStepAdvance)) AND NOT #bOutEnterEvent) THEN 
               #iCurrentStep   := #iInNextStep;   //move to next step
               //Reset Step done Timer
               #TON_StepDelay(IN:=(false),PT:=#tInStepDelay); 
               #bOutExitEvent:=true;
               #bAlreadyInThisStep:=false;
           END_IF;
       END_IF;
       #bOutPaused := #bInStepDone AND (#TON_StepDelay.Q OR #bNoStepDelay) AND (#bInStepMode AND NOT #bInStepAdvance);
       //Only set this if we are ok and in the right step
       ENO:= true;
   END_IF;
   IF (#bInit) THEN
       #iCurrentStep := #iInitStep;
       #bInit:=false;  //Clear so that if it is unwired on the next call, it is not run.
       #bAlreadyInThisStep:=false;
   END_IF;

   //Set output variables
   #iOutCurrentStep := #iCurrentStep;
   #tInStepDelay := T#0MS;
END_FUNCTION_BLOCK

FUNCTION "fcStepChooser" : Int   // FC185, SCL
{ S7_Optimized_Access := 'TRUE' }
VERSION : 0.0
   VAR_INPUT
      bCondition : Bool;
      iTrueStep : Int;
      iFalseStep : Int;
   END_VAR
   VAR_TEMP
      iResult : Int;
   END_VAR
BEGIN

       IF #bCondition THEN
           #iResult:=#iTrueStep;
       ELSE
           #iResult:=#iFalseStep;
       END_IF;
       ENO:=true;
       #fcStepChooser:=#iResult;
END_FUNCTION

// folder: Open Library V15/Resources/HMI

FUNCTION_BLOCK "fbErrorScroller"   // FB330, FBD
TITLE = Scrolls through the error codes for display on the HMI
{ S7_Optimized_Access := 'TRUE' }
AUTHOR : DMC
FAMILY : Error
VERSION : 0.1
   VAR_INPUT
      bInError01 : Bool;   // Error 1 In Error Array
      bInError02 : Bool;   // Error 2 In Error Array
      bInError03 : Bool;   // Error 3 In Error Array
      bInError04 : Bool;   // Error 4 In Error Array
      bInError05 : Bool;   // Error 5 In Error Array
      bInError06 : Bool;   // Error 6 In Error Array
      bInError07 : Bool;   // Error 7 In Error Array
      bInError08 : Bool;   // Error 8 In Error Array
      bInError09 : Bool;   // Error 9 In Error Array
      bInError10 : Bool;   // Error 10 In Error Array
      bInError11 : Bool;   // Error 11 In Error Array
      bInError12 : Bool;   // Error 12 In Error Array
      bInError13 : Bool;   // Error 13 In Error Array
      bInError14 : Bool;   // Error 14 In Error Array
      bInError15 : Bool;   // Error 15 In Error Array
      bInError16 : Bool;   // Error 16 In Error Array
      bInError17 : Bool;   // Error 17 In Error Array
      bInError18 : Bool;   // Error 18 In Error Array
      bInError19 : Bool;   // Error 19 In Error Array
      bInError20 : Bool;   // Error 20 In Error Array
      bInError21 : Bool;   // Error 21 In Error Array
      bInError22 : Bool;   // Error 22 In Error Array
      bInError23 : Bool;   // Error 23 In Error Array
      bInError24 : Bool;   // Error 24 In Error Array
      bInError25 : Bool;   // Error 25 In Error Array
      bInError26 : Bool;   // Error 26 In Error Array
      bInError27 : Bool;   // Error 27 In Error Array
      bInError28 : Bool;   // Error 28 In Error Array
      bInError29 : Bool;   // Error 29 In Error Array
      bInError30 : Bool;   // Error 30 In Error Array
   END_VAR
   VAR_OUTPUT
      bOutErrorExists : Bool;   // An Error Exists
      iOutScrollingErrorNumber : Int;   // Current Index when scrolling through errors
   END_VAR
   VAR
      TON_ErrorDelay : TON_TIME;   // Delay between each scroll for a new error
      abErrors : Array[#ciIndexLow..#ciIndexHigh] of Bool;
      iNextScrollNum : Int := 1;   // Index of next error position
      iErrorsScrollNum : Int := 1;   // Index of current error position
      bScrolling : Bool;   // Indicates we are scrolling
      bTON_ErrorDelay : Bool;
   END_VAR
   VAR_TEMP
      bErrorExists : Bool;   // Error Exists
   END_VAR
   VAR CONSTANT
      ciNoErrrors : Int := 0;
      ciIndexLow : Int := 1;
      ciIndexHigh : Int := 30;
   END_VAR
   VAR_TEMP   // added for the SCL form of the ladder/FBD networks
      _w1 : Bool;
   END_VAR
BEGIN

REGION Network 1: Check for valid array indexes
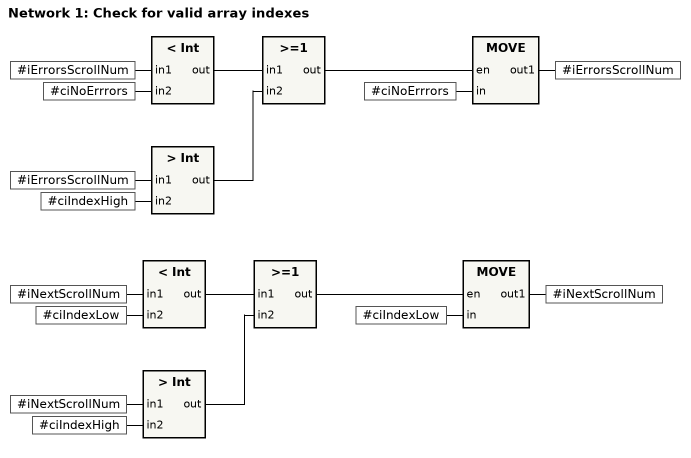
   IF (#iErrorsScrollNum < #ciNoErrrors) OR (#iErrorsScrollNum > #ciIndexHigh) THEN
       #iErrorsScrollNum := #ciNoErrrors;
   END_IF;
   IF (#iNextScrollNum < #ciIndexLow) OR (#iNextScrollNum > #ciIndexHigh) THEN
       #iNextScrollNum := #ciIndexLow;
   END_IF;
END_REGION

REGION Network 2: Check if error exists
   // OR all of the possible errors. If any error Exists, SET bErrorExists
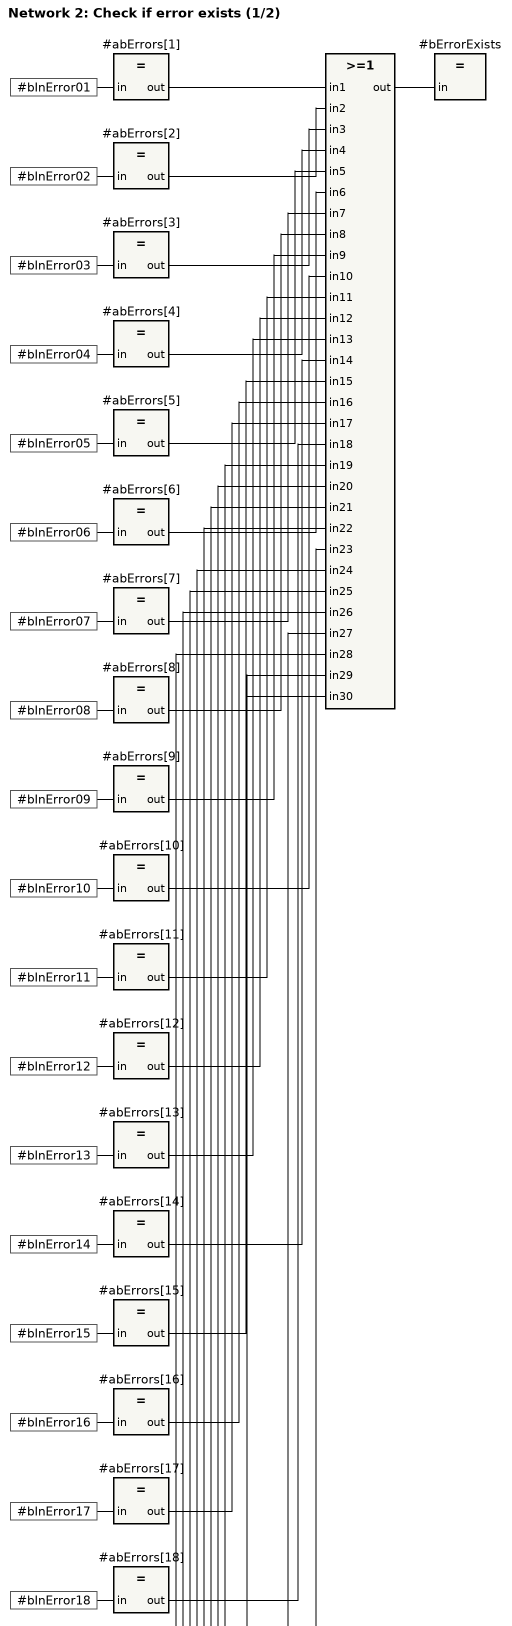
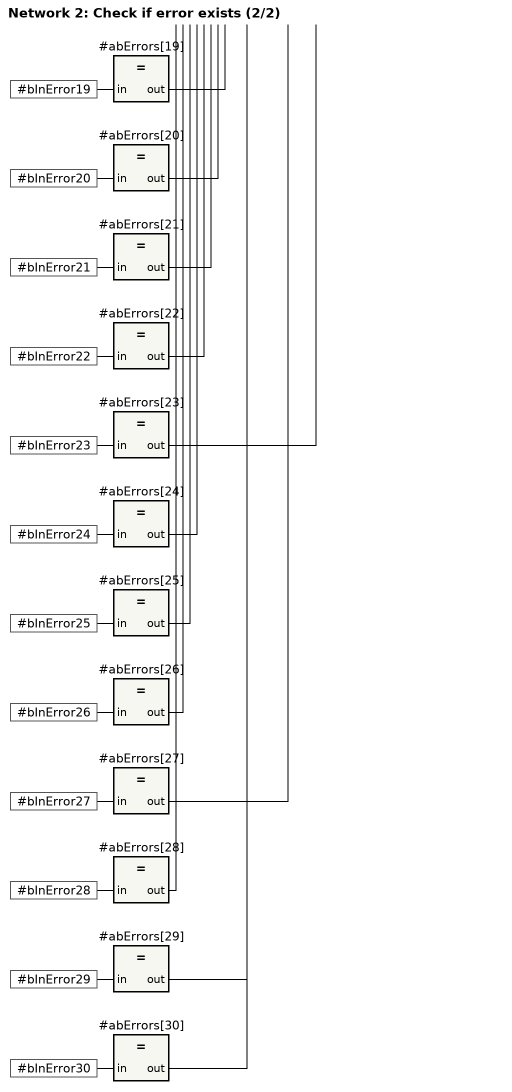
   #abErrors[1] := #bInError01;
   #abErrors[2] := #bInError02;
   #abErrors[3] := #bInError03;
   #abErrors[4] := #bInError04;
   #abErrors[5] := #bInError05;
   #abErrors[6] := #bInError06;
   #abErrors[7] := #bInError07;
   #abErrors[8] := #bInError08;
   #abErrors[9] := #bInError09;
   #abErrors[10] := #bInError10;
   #abErrors[11] := #bInError11;
   #abErrors[12] := #bInError12;
   #abErrors[13] := #bInError13;
   #abErrors[14] := #bInError14;
   #abErrors[15] := #bInError15;
   #abErrors[16] := #bInError16;
   #abErrors[17] := #bInError17;
   #abErrors[18] := #bInError18;
   #abErrors[19] := #bInError19;
   #abErrors[20] := #bInError20;
   #abErrors[21] := #bInError21;
   #abErrors[22] := #bInError22;
   #abErrors[23] := #bInError23;
   #abErrors[24] := #bInError24;
   #abErrors[25] := #bInError25;
   #abErrors[26] := #bInError26;
   #abErrors[27] := #bInError27;
   #abErrors[28] := #bInError28;
   #abErrors[29] := #bInError29;
   #abErrors[30] := #bInError30;
   #bErrorExists := #bInError01 OR #bInError02 OR #bInError03 OR #bInError04 OR #bInError05 OR #bInError06 OR #bInError07 OR #bInError08 OR #bInError09 OR #bInError10 OR #bInError11 OR #bInError12 OR #bInError13 OR #bInError14 OR #bInError15 OR #bInError16 OR #bInError17 OR #bInError18 OR #bInError19 OR #bInError20 OR #bInError21 OR #bInError22 OR #bInError23 OR #bInError24 OR #bInError25 OR #bInError26 OR #bInError27 OR #bInError28 OR #bInError29 OR #bInError30;
END_REGION

REGION Network 3: Timer to change displayed error
   // ============================ Scroll errors on HMI ========================
   // Timed delay
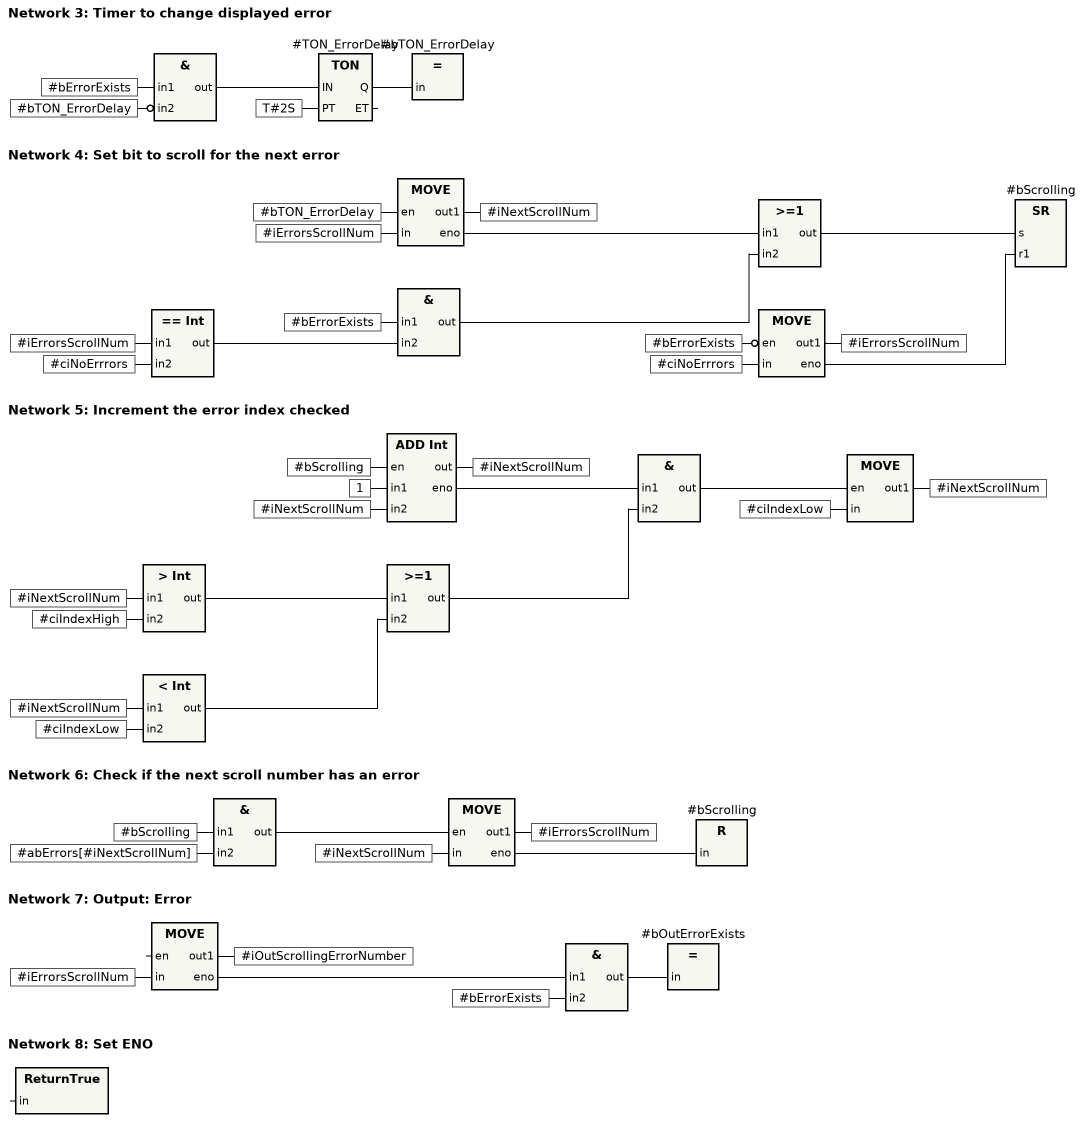
   #TON_ErrorDelay(IN := #bErrorExists AND NOT #bTON_ErrorDelay, PT := T#2S);   // TON
   #bTON_ErrorDelay := #TON_ErrorDelay.Q;
END_REGION

REGION Network 4: Set bit to scroll for the next error
   // Set a static bit indicating that we are scrolling.  
   // Each pass cycle through the function, we will increment.  
   // If there is no error, set the scroll num to 0 and turn off scrolling.  
   // It scrolls to an error immediately when an error occurs.
   // ENO of a box is taken as its EN; it also drops when the box reports an error
   IF #bTON_ErrorDelay THEN #iNextScrollNum := #iErrorsScrollNum; END_IF;
   #_w1 := #bTON_ErrorDelay OR (#bErrorExists AND (#iErrorsScrollNum = #ciNoErrrors));
   IF NOT #bErrorExists THEN #iErrorsScrollNum := #ciNoErrrors; END_IF;
   IF #_w1 THEN
       #bScrolling := TRUE;   // SR flip-flop
   END_IF;
   IF NOT #bErrorExists THEN #bScrolling := FALSE; END_IF;
END_REGION

REGION Network 5: Increment the error index checked
   // The function will only increment the scroll num one value per scan.  
   // It will scroll until it finds the next active error, then stop scrolling.  
   // Roll iNextScrollNum to 0 if it exceeds 30.
   // ENO of a box is taken as its EN; it also drops when the box reports an error
   IF #bScrolling THEN #iNextScrollNum := 1 + #iNextScrollNum; END_IF;
   IF #bScrolling AND ((#iNextScrollNum > #ciIndexHigh) OR (#iNextScrollNum < #ciIndexLow)) THEN
       #iNextScrollNum := #ciIndexLow;
   END_IF;
END_REGION

REGION Network 6: Check if the next scroll number has an error
   // If we found an error, stop scrolling.
   // ENO of a box is taken as its EN; it also drops when the box reports an error
   IF #bScrolling AND #abErrors[#iNextScrollNum] THEN
       #iErrorsScrollNum := #iNextScrollNum;
       #bScrolling := FALSE;
   END_IF;
END_REGION

REGION Network 7: Output: Error
   // Output the index of the error that exists.
   // ENO of a box is taken as its EN; it also drops when the box reports an error
   #iOutScrollingErrorNumber := #iErrorsScrollNum;
   #bOutErrorExists := #bErrorExists;
END_REGION

REGION Network 8: Set ENO
   ENO := TRUE;
   RETURN;
END_REGION
END_FUNCTION_BLOCK

FUNCTION "fcHMIBitEnable" : Void   // FC329, FBD
TITLE = Handles an async reading of an HMI bit to avoid race conditions, includes an enable bit
{ S7_Optimized_Access := 'TRUE' }
VERSION : 0.1
   VAR_INPUT
      bInToggle : Bool;
      bInLatch : Bool;
      bInEnable : Bool;
   END_VAR
   VAR_OUTPUT
      bOutEnable : Bool;
   END_VAR
   VAR_IN_OUT
      bInOutHMI : Bool;
      bInOutPLC : Bool;
   END_VAR
   VAR_TEMP   // added for the SCL form of the ladder/FBD networks
      _w1 : Bool;
   END_VAR
BEGIN

REGION Network 1: If not latching or toggling, reset the PLC bit every scan
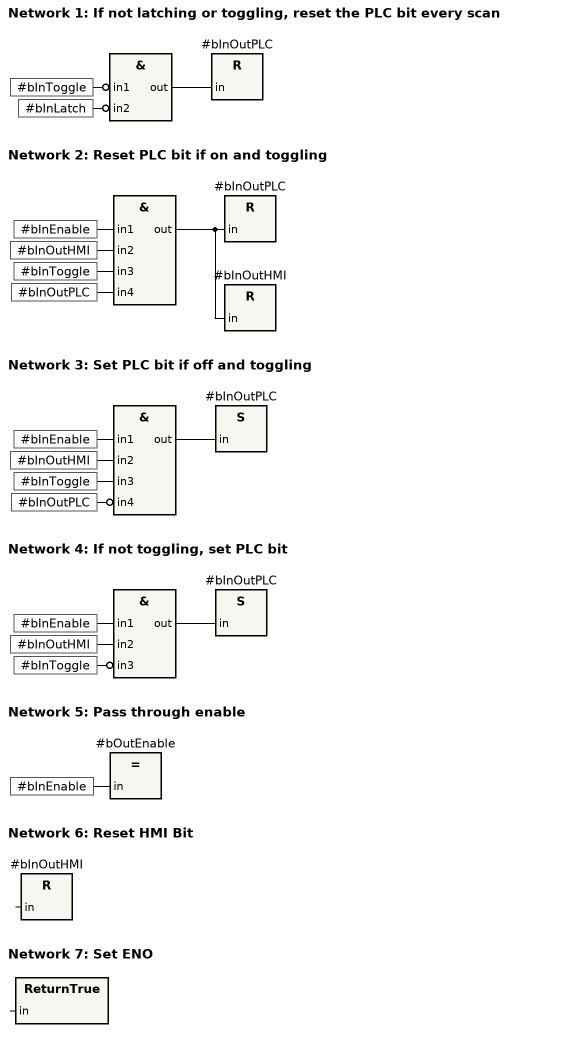
   IF NOT #bInToggle AND NOT #bInLatch THEN #bInOutPLC := FALSE; END_IF;
END_REGION

REGION Network 2: Reset PLC bit if on and toggling
   #_w1 := #bInEnable AND #bInOutHMI AND #bInToggle AND #bInOutPLC;
   IF #_w1 THEN
       #bInOutPLC := FALSE;
       #bInOutHMI := FALSE;
   END_IF;
END_REGION

REGION Network 3: Set PLC bit if off and toggling
   IF #bInEnable AND #bInOutHMI AND #bInToggle AND NOT #bInOutPLC THEN #bInOutPLC := TRUE; END_IF;
END_REGION

REGION Network 4: If not toggling, set PLC bit
   IF #bInEnable AND #bInOutHMI AND NOT #bInToggle THEN #bInOutPLC := TRUE; END_IF;
END_REGION

REGION Network 5: Pass through enable
   #bOutEnable := #bInEnable;
END_REGION

REGION Network 6: Reset HMI Bit
   #bInOutHMI := FALSE;
END_REGION

REGION Network 7: Set ENO
   ENO := TRUE;
   RETURN;
END_REGION
END_FUNCTION

FUNCTION "fcSetHMIStatusSimulation" : Void   // FC333, FBD
TITLE = Sets HMI Status
{ S7_Optimized_Access := 'TRUE' }
VERSION : 0.1
// Wrapper function for setting the HMI status of a device
// 
// In order of priority:
// 1. E-stop
// 2. Error
// 3. Forward/Work Position
// 4. Reverse/Home Position
// 5. Forward/Work On
// 6. Reverse/Home On
// 7. None
   VAR_INPUT
      bInEstop : Bool;
      bInError : Bool;
      bInForwardWork : Bool;
      bInReverseHome : Bool;
      bInOnForwardWork : Bool;
      bInOnReverseHome : Bool;
      bInSimulate : Bool;
   END_VAR
   VAR_OUTPUT
      iOutStatus : Int;
   END_VAR
BEGIN

REGION Network 1: Set Reverse/Home On
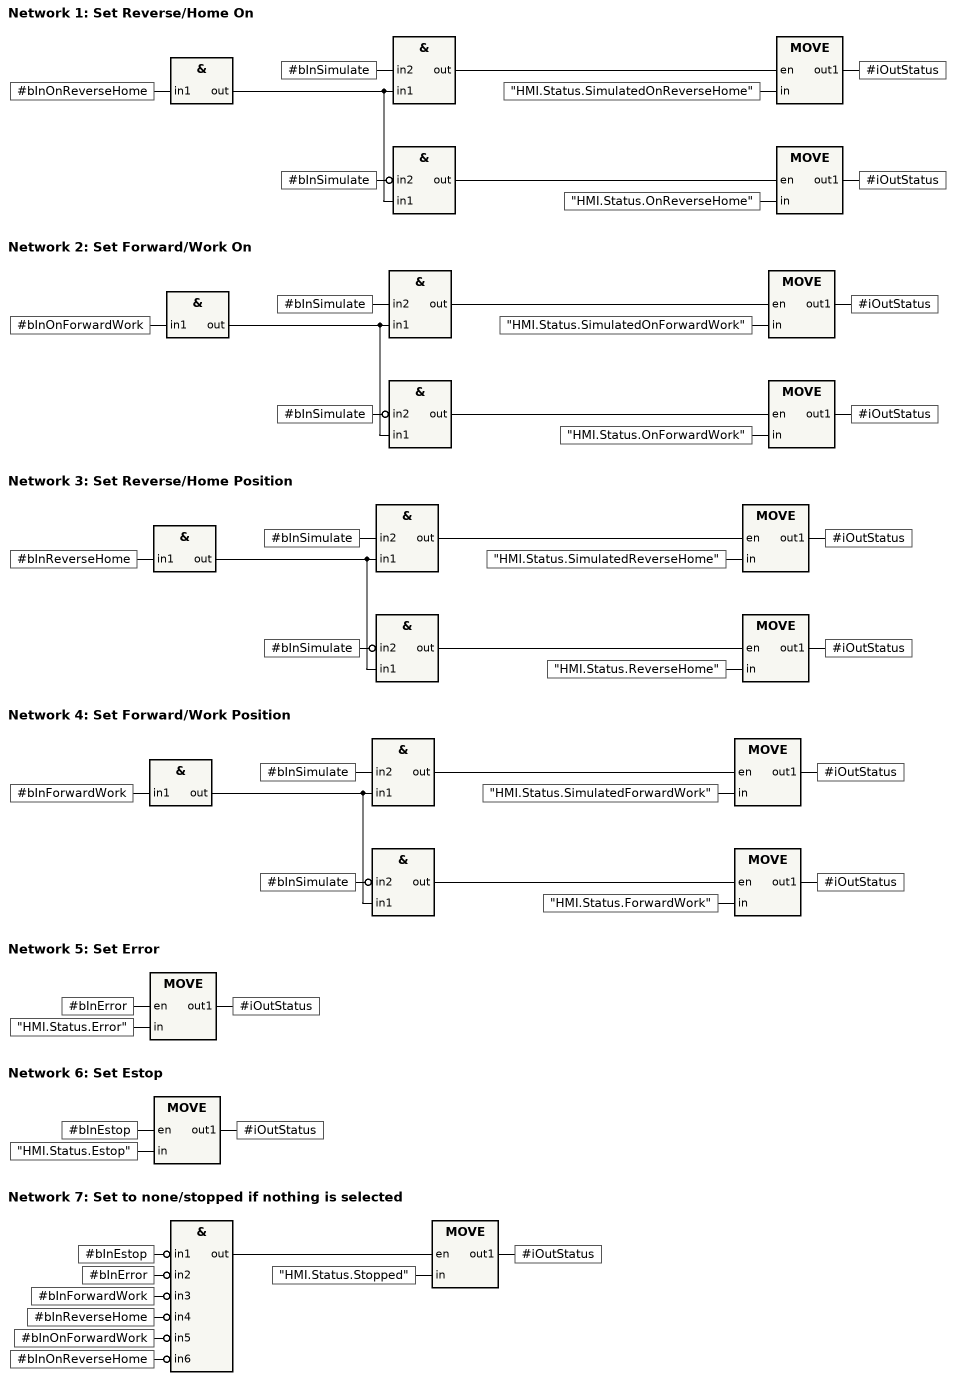
   IF #bInSimulate AND #bInOnReverseHome THEN #iOutStatus := "HMI.Status.SimulatedOnReverseHome"; END_IF;
   IF NOT #bInSimulate AND #bInOnReverseHome THEN #iOutStatus := "HMI.Status.OnReverseHome"; END_IF;
END_REGION

REGION Network 2: Set Forward/Work On
   IF #bInSimulate AND #bInOnForwardWork THEN #iOutStatus := "HMI.Status.SimulatedOnForwardWork"; END_IF;
   IF NOT #bInSimulate AND #bInOnForwardWork THEN #iOutStatus := "HMI.Status.OnForwardWork"; END_IF;
END_REGION

REGION Network 3: Set Reverse/Home Position
   IF #bInSimulate AND #bInReverseHome THEN #iOutStatus := "HMI.Status.SimulatedReverseHome"; END_IF;
   IF NOT #bInSimulate AND #bInReverseHome THEN #iOutStatus := "HMI.Status.ReverseHome"; END_IF;
END_REGION

REGION Network 4: Set Forward/Work Position
   IF #bInSimulate AND #bInForwardWork THEN #iOutStatus := "HMI.Status.SimulatedForwardWork"; END_IF;
   IF NOT #bInSimulate AND #bInForwardWork THEN #iOutStatus := "HMI.Status.ForwardWork"; END_IF;
END_REGION

REGION Network 5: Set Error
   IF #bInError THEN #iOutStatus := "HMI.Status.Error"; END_IF;
END_REGION

REGION Network 6: Set Estop
   IF #bInEstop THEN #iOutStatus := "HMI.Status.Estop"; END_IF;
END_REGION

REGION Network 7: Set to none/stopped if nothing is selected
   IF NOT #bInEstop AND NOT #bInError AND NOT #bInForwardWork AND NOT #bInReverseHome AND NOT #bInOnForwardWork AND NOT #bInOnReverseHome THEN
       #iOutStatus := "HMI.Status.Stopped";
   END_IF;
END_REGION

REGION Network 8: Set ENO
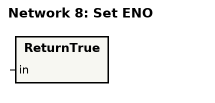
   ENO := TRUE;
   RETURN;
END_REGION
END_FUNCTION

// folder: TestBlocks

FUNCTION_BLOCK "TestExecOrd2"   // FB6, FBD
{ S7_Optimized_Access := 'TRUE' }
VERSION : 0.1
BEGIN

REGION Network 1: X != 10
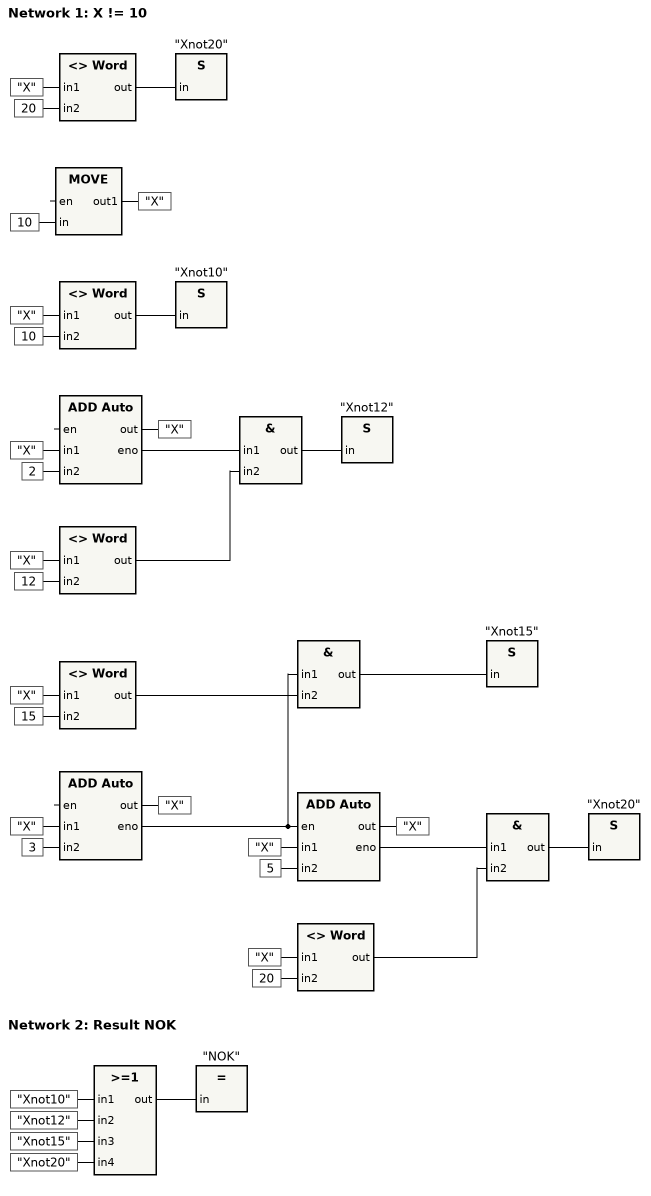
   IF "X" <> 20 THEN "Xnot20" := TRUE; END_IF;
   "X" := 10;
   IF "X" <> 10 THEN "Xnot10" := TRUE; END_IF;
   "X" := "X" + 2;
   IF "X" <> 12 THEN "Xnot12" := TRUE; END_IF;
   "X" := "X" + 3;
   IF "X" <> 15 THEN "Xnot15" := TRUE; END_IF;
   "X" := "X" + 5;
   IF "X" <> 20 THEN "Xnot20" := TRUE; END_IF;
END_REGION

REGION Network 2: Result NOK
   "NOK" := "Xnot10" OR "Xnot12" OR "Xnot15" OR "Xnot20";
END_REGION

REGION Network 3: Result NOK
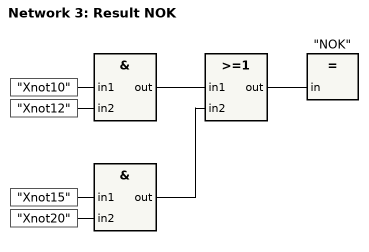
   "NOK" := ("Xnot10" AND "Xnot12") OR ("Xnot15" AND "Xnot20");
END_REGION
END_FUNCTION_BLOCK

FUNCTION "TestExecOrd" : Void   // FC2, FBD
{ S7_Optimized_Access := 'TRUE' }
VERSION : 0.1
BEGIN

REGION Network 1
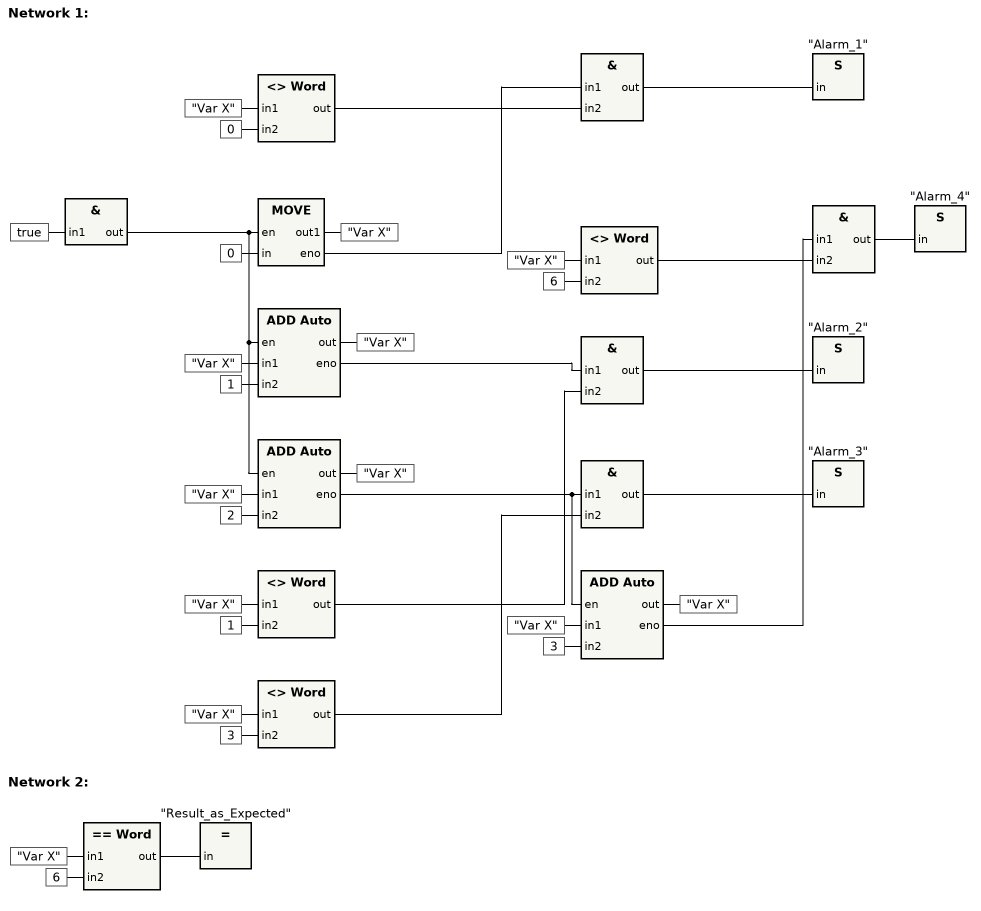
   IF true THEN "Var X" := 0; END_IF;
   IF true AND ("Var X" <> 0) THEN "Alarm_1" := TRUE; END_IF;
   IF true THEN "Var X" := "Var X" + 1; END_IF;
   IF true AND ("Var X" <> 1) THEN "Alarm_2" := TRUE; END_IF;
   IF true THEN "Var X" := "Var X" + 2; END_IF;
   IF true AND ("Var X" <> 3) THEN "Alarm_3" := TRUE; END_IF;
   IF true THEN "Var X" := "Var X" + 3; END_IF;
   IF true AND ("Var X" <> 6) THEN "Alarm_4" := TRUE; END_IF;
END_REGION

REGION Network 2
   "Result_as_Expected" := "Var X" = 6;
END_REGION
END_FUNCTION

// ===== library: MasterCopy "Block_FBD" =====

FUNCTION "Block_FBD" : Void   // FC3, FBD
{ S7_Optimized_Access := 'FALSE' }
VERSION : 0.1
BEGIN
END_FUNCTION

// ===== library: MasterCopy "Block_LAD" =====

FUNCTION "Block_LAD" : Void   // FC2, LAD
{ S7_Optimized_Access := 'FALSE' }
VERSION : 0.1
BEGIN
END_FUNCTION

// ===== library: MasterCopy "Block_SCL" =====

FUNCTION "Block_SCL" : Void   // FC5, SCL
{ S7_Optimized_Access := 'FALSE' }
VERSION : 0.1
BEGIN
END_FUNCTION

// ===== library: MasterCopy "Block_STL" =====

FUNCTION "Block_STL" : Void   // FC4, STL
{ S7_Optimized_Access := 'FALSE' }
VERSION : 0.1
BEGIN
END_FUNCTION